FUNCTION_BLOCK AnalogInput_Standard EXTENDS AnalogInput IMPLEMENTS I_AnalogChannel_Standard
VAR
	Status : REFERENCE TO ST_AnalogInputStatus_EL30xx;
END_VAR

PROPERTY DataValid : BOOL
GET
DataValid := NOT Status.TxPDOState;
END_GET
END_PROPERTY

PROPERTY Error : BOOL
GET
Error := Status.Error;
END_GET
END_PROPERTY

(*FB_Init is always available implicitly and it is used primarily for initialization.
The return value is not evaluated. For a specific influence, you can also declare the
methods explicitly and provide additional code there with the standard initialization
code. You can evaluate the return value.*)
METHOD FB_Init : BOOL
VAR_INPUT
	(* TRUE: the retain variables are initialized (reset warm / reset cold)*)
	bInitRetains : BOOL;

	(* TRUE: the instance will be copied to the copy code afterward (online change)   *)
	bInCopyCode : BOOL;
	Name		: T_MaxString;
	Input		: REFERENCE TO INT;
	Status		: REFERENCE TO ST_AnalogInputStatus_EL30xx;
END_VAR
THIS^.Status REF= Status;
END_METHOD

PROPERTY Limit1High : BOOL
GET
Limit1High := Status.Limit1H;
END_GET
END_PROPERTY

PROPERTY Limit1Low : BOOL
GET
Limit1Low := Status.Limit1L;
END_GET
END_PROPERTY

PROPERTY Limit2High : BOOL
GET
Limit2High := Status.Limit2H;
END_GET
END_PROPERTY

PROPERTY Limit2Low : BOOL
GET
Limit2Low := Status.Limit2L;
END_GET
END_PROPERTY

PROPERTY Overrange : BOOL
GET
Overrange := Status.Overrange;
END_GET
END_PROPERTY

PROPERTY Underrange : BOOL
GET
Underrange := Status.Underrrange;
END_GET
END_PROPERTY

END_FUNCTION_BLOCK

(* stored: Version 1.1.0.1, ProductVersion 3.1.4026.18
   POU AnalogInput_Standard: Id {71805f60-3fa6-4837-90c8-ebd868d11a17}, SpecialFunc None
   Property DataValid: Id {c9db11b9-c3d3-49c3-9ee1-33b16d646fe1}
   Get Get: Id {c668b64a-efdd-478e-bd92-5ac1f8eefa15}
   Property Error: Id {13dc8754-b7ef-4c4f-8726-89334a7e4ddd}
   Get Get: Id {759954c3-60f4-47c6-9804-6581331863eb}
   Method FB_Init: Id {da7ffb6f-59a5-4357-8511-56879d963281}
   Property Limit1High: Id {e68c18bb-9f09-48b4-9a9d-286a6fa63815}
   Get Get: Id {b4c3c05d-7590-4ed6-b0fe-79488f13ed29}
   Property Limit1Low: Id {f50fcef9-2071-493b-a192-2134686ea5ee}
   Get Get: Id {82881d7e-67d6-43b0-bbc5-14854e78125e}
   Property Limit2High: Id {9ecc57d7-603e-447f-aa1e-4bc207f30ea5}
   Get Get: Id {82719071-2c7e-449b-9161-2c6d62cb5882}
   Property Limit2Low: Id {02101e3a-1ef3-4e7e-8a38-278050a16640}
   Get Get: Id {7bb4c7df-1d9f-47dd-8da5-875ca72c29d5}
   Property Overrange: Id {3453a052-5e78-41c4-b6e2-7b4479cb77da}
   Get Get: Id {8a53c3f0-6fe1-4492-b624-03d328d0b792}
   Property Underrange: Id {cf676880-ef4a-4f10-91e9-838c4db84b1d}
   Get Get: Id {2c4e6e30-5aef-4444-877a-0d7d4e57f9e4} *)
